// TwinCAT 3 PLC project Test_Project
// ProgramVersion: 3.1.4024.0
// libraries:
//   Project_Logic_1, * (InTimeTec)
//   Tc2_Standard, * (Beckhoff Automation GmbH)
//   Tc2_System, * (Beckhoff Automation GmbH)
//   Tc3_Module, * (Beckhoff Automation GmbH)
//   TcUnit, * (www.tcunit.org)
// project tree:
//   / PlcTask.TcTTO
//   POUs/ PRG_TEST.TcPOU
//   TESTs/ FB_BottleFiller_Test.TcPOU
// real-time tasks:
//   TASK PlcTask: cycle T#10ms, priority 20, ADS port 350
//   TASK PlcTask1: cycle T#10ms, priority 21, ADS port 351

CONFIGURATION Test_Project
    RESOURCE PLC ON TwinCAT3
        TASK PlcTask(INTERVAL := T#10ms, PRIORITY := 20);
        PROGRAM PRG_TEST WITH PlcTask : PRG_TEST;
    END_RESOURCE
END_CONFIGURATION

// ---- POUs/PRG_TEST.TcPOU
PROGRAM PRG_TEST
VAR
	
fbBottleFiller_Test : FB_BottleFiller_Test;
fbBottle : FB_BottleFiller;
END_VAR


TcUnit.RUN();

END_PROGRAM

// ---- TESTs/FB_BottleFiller_Test.TcPOU
FUNCTION_BLOCK FB_BottleFiller_Test EXTENDS FB_TestSuite

VAR	
END_VAR

TurningOnTheValveIfValveIsEmpty();

METHOD SettingThePressure
VAR_INPUT
END_VAR
END_METHOD

METHOD TurningOnTheValveIfValveIsEmpty
VAR_INPUT
END_VAR
VAR
	fbBottleFiller : FB_BottleFiller;
	fbBottle : FB_BottleFiller;
END_VAR
TEST('TurningOnTheValveIfValveIsEmpty');

fbBottleFiller.bisTankEmpty := TRUE;
fbBottleFiller.StartFilling();
AssertTrue(Condition := fbBottleFiller.bFilling,
		   Message := 'Tank is not Empty');

fbBottleFiller.bLevelSensor := TRUE;
fbBottleFiller.StopFilling();

AssertFalse(Condition := fbBottleFiller.bFilling, 
			 Message := 'Tank is filling');
TEST_FINISHED();
END_METHOD

END_FUNCTION_BLOCK
